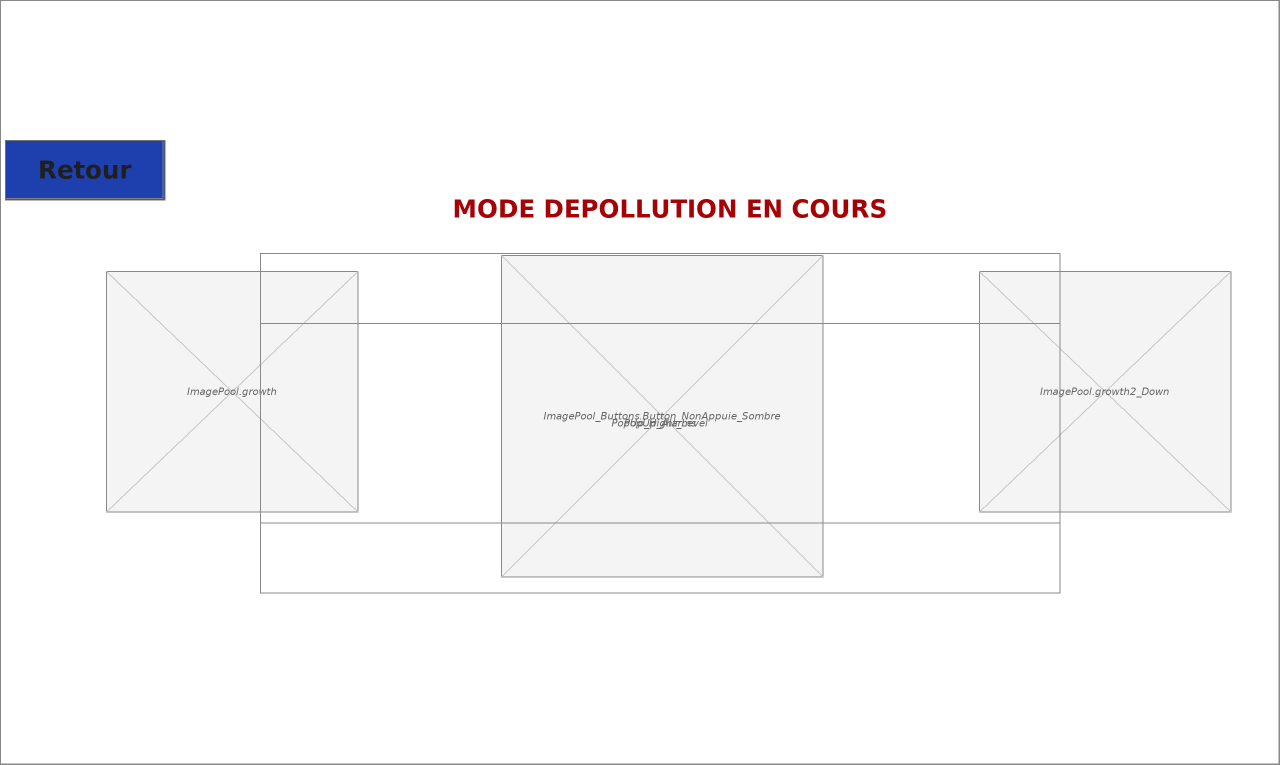
VISUALIZATION Depollution  // 1280x765
    Frame (0,0 1280x765)
        shows masque()
    Button (5,140 160x60), "Retour", invisible if: Mode_Cabine_Depollution
        OnMouseDown: change screen: menu
    Image (501,255 322x322), image: ImagePool_Buttons.Button_Appuie_Sombre
    Image (501,255 322x322), invisible if: Start_Etat_Depollution, image: ImagePool_Buttons.Button_NonAppuie_Sombre
        OnMouseDown: toggle Start_Etat_Depollution
    Image (106,271 252x241), image: ImagePool.growth
        p2738717112: GVL_Visu.Arrow_Up
    Image (979,271 252x241), image: ImagePool.growth2_Down
        p2738717112: GVL_Visu.Arrow_Down
    Rectangle (106,214 252x50), "EXTRACTION"
    Rectangle (979,214 252x50), "SOUFFLAGE"
    Group (265,185 809x545), invisible if: NOT Mode_Cabine_Depollution
        Rectangle (81,0 648x48), "MODE DEPOLLUTION EN COURS", invisible if: GVL_Visu.On_Off_Anim
        Group (0,497 809x48)
            Rectangle (0,0 315x48), "%.0f heure(s)", text variable: Lect_Temp_heure_Depol, invisible if: NOT Mode_Cabine_Depollution
            Rectangle (318,0 220x48), "%.0f minute(s)", text variable: Lect_Temp_Minute_Depol, invisible if: NOT Mode_Cabine_Depollution
            Rectangle (530,0 279x48), "%.0f seconde(s)", text variable: Lect_Temp_Seconde_Depol, invisible if: NOT Mode_Cabine_Depollution
    Rectangle (444,586 451x48), "Consigne : %.0f Vol/h", text variable: Cons_Deb_Souf_Etat_Depol
    Rectangle (444,634 451x48), "Mesure : %.0f Vol/h", text variable: Visu.IHM_Mesure_Debit_Deconta
    Group (420,683 500x64), invisible if: Mode_Cabine_Depollution
        RoundedRectangle (0,0 237x64), "%.0f heure(s)", text variable: Cons_Temp_heure_Depol
            OnMouseDown: write the text variable via VisuDialogs.Numpad, min 0, max 23, format %.0f
        RoundedRectangle (237,0 263x64), "%.0f minute(s)", text variable: Cons_Temp_Minute_Depol
            OnMouseDown: write the text variable via VisuDialogs.Numpad, min 0, max 59, format %.0f
    Group (260,253 800x340)
        Frame (0,0 800x340), invisible if: NOT GVL_Visu.Affichage_PopUp_Alarm
            shows PopUp_Alarms()
        Frame (0,70 800x200), invisible if: NOT GVL_Visu.Affichage_PopUp_HightLevel
            shows PopUp_Hight_Level()
END_VISUALIZATION

(* stored: Version 1.1.0.1, ProductVersion 3.1.4024.16
   Visu Depollution: Id {0e9504e9-9485-4a58-89a2-41947f428448} *)
